TYPE RemoteFeedbackStewart :
STRUCT
	surge : REAL;
	sway : REAL;
	heave : REAL;
	phi : REAL;
	theta : REAL;
	psi	: REAL;
	surge_t	: REAL;
	sway_t	: REAL;
	heave_t	: REAL;
	wx : REAL;
	wy : REAL;
	wz : REAL;
	surge_tt : REAL;
	sway_tt : REAL;
	heave_tt : REAL;
	wx_t	: REAL;
	wy_t : REAL;
	wz_t : REAL;
END_STRUCT
END_TYPE

(* stored: Version 1.1.0.1, ProductVersion 3.1.4020.12
   DUT RemoteFeedbackStewart: Id {dbe9f13a-90b3-482d-a35b-3c357fc25569} *)
